FUNCTION_BLOCK FB_NTZ
VAR_INPUT
END_VAR
VAR_OUTPUT
END_VAR
VAR
	Kaltwasser_1xx	: FB_NTZ_KW;
	Warmwasser_2xx	: FB_NTZ_WW;
	Heisswasser_3xx	: FB_NTZ_HW;
	{attribute 'OPC.UA.DA' := '1'}Freigabe_KW		: BOOL :=TRUE; 
	{attribute 'OPC.UA.DA' := '1'}Freigabe_WW		: BOOL :=TRUE; 
	{attribute 'OPC.UA.DA' := '1'}Freigabe_HW		: BOOL :=TRUE; 
	DS_100_KWN				: FB_DS;
	DS_200_WWN				: FB_DS;
	DS_300_HWN				: FB_DS;

END_VAR

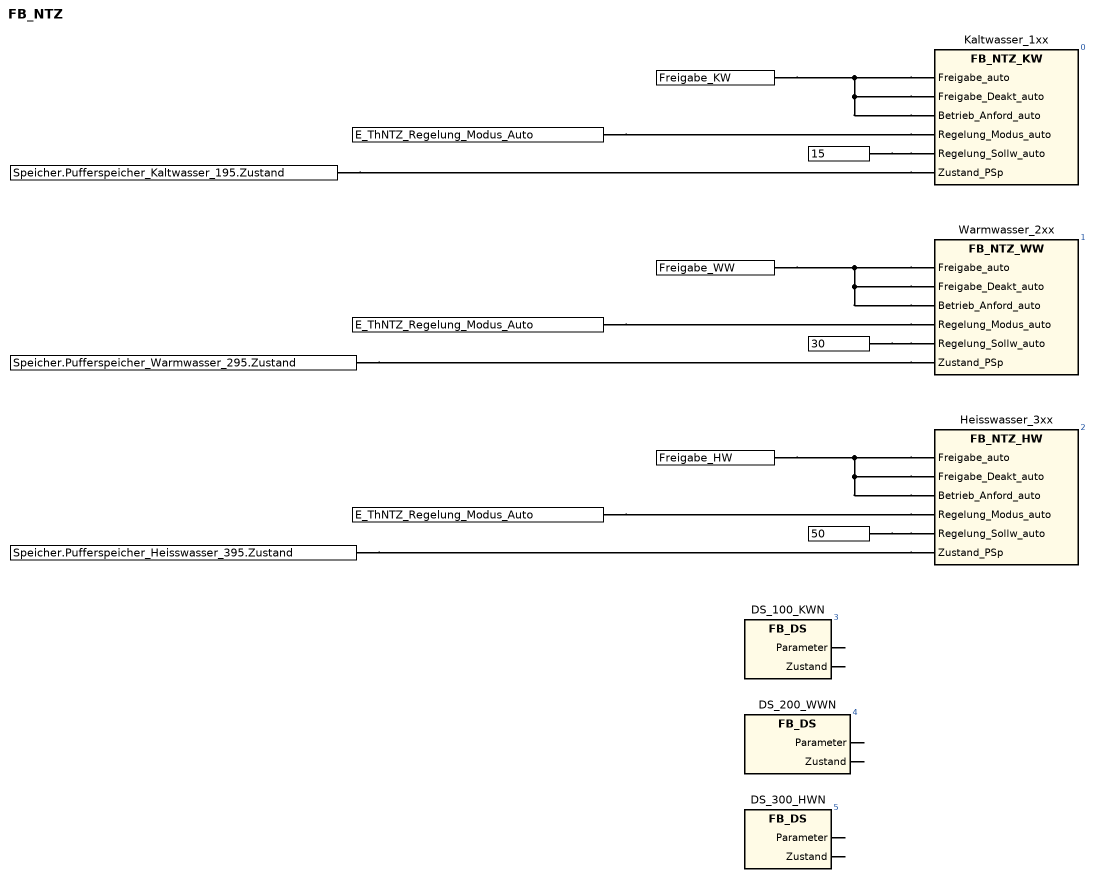
Kaltwasser_1xx(
    Freigabe_auto := Freigabe_KW,
    Freigabe_Deakt_auto := Freigabe_KW,
    Betrieb_Anford_auto := Freigabe_KW,
    Regelung_Modus_auto := E_ThNTZ_Regelung_Modus_Auto,
    Regelung_Sollw_auto := 15,
    Zustand_PSp := Speicher.Pufferspeicher_Kaltwasser_195.Zustand); // FB_NTZ_KW
Warmwasser_2xx(
    Freigabe_auto := Freigabe_WW,
    Freigabe_Deakt_auto := Freigabe_WW,
    Betrieb_Anford_auto := Freigabe_WW,
    Regelung_Modus_auto := E_ThNTZ_Regelung_Modus_Auto,
    Regelung_Sollw_auto := 30,
    Zustand_PSp := Speicher.Pufferspeicher_Warmwasser_295.Zustand); // FB_NTZ_WW
Heisswasser_3xx(
    Freigabe_auto := Freigabe_HW,
    Freigabe_Deakt_auto := Freigabe_HW,
    Betrieb_Anford_auto := Freigabe_HW,
    Regelung_Modus_auto := E_ThNTZ_Regelung_Modus_Auto,
    Regelung_Sollw_auto := 50,
    Zustand_PSp := Speicher.Pufferspeicher_Heisswasser_395.Zustand); // FB_NTZ_HW
DS_100_KWN(); // FB_DS
DS_200_WWN(); // FB_DS
DS_300_HWN(); // FB_DS

END_FUNCTION_BLOCK

(* stored: Version 1.1.0.1, ProductVersion 3.1.4024.9
   POU FB_NTZ: Id {46d1b285-671a-4902-a14c-ef9407c9bc7e}, SpecialFunc None *)
